// TIA Portal project "Smith Predictor Controller 20211018" (V15.1)

(* hardware
DEVICE "S71500/ET200MP station_1"  S7-1500 station
   slot 0: "导轨_0"  Rack  6ES7 590-1***0-0AA0
   slot 1: "PLC_1"  CPU 1516-3 PN/DP  6ES7 516-3AN01-0AB0  V2.6
      slot 3: "CPU 显示_1"  6ES7591-1BA00-0AA0
*)

// ===== PLC "PLC_1"  CPU 1516-3 PN/DP =====

// folder: smith

DATA_BLOCK "SIM_DB"   // DB1
{ S7_Optimized_Access := 'TRUE' }
VERSION : 0.1
   VAR
      SIM_RUN : Bool;
      PLANT_PV_SMITH : Real;
      PLANT_PV_PID : Real;
      "PLANT_TAU_ACTUAL[ms]" : Real := 500.0;
      "PLANT_DELAY_ACTUAL[Ncycle]" : Int := 50;
      "PLANT_TAU_SET[ms]" : Real := 500.0;
      PLANT_TAU_SET_MIN : Real := 475.0;
      PLANT_TAU_SET_MAX : Real := 525.0;
      "PLANT_DELAY_SET[s]" : Real := 5.0;
      "PLANT_DELAY_SET[Ncycle]" : Int := 50;
      PLANT_DELAY_SET_MIN : Int := 45;
      PLANT_DELAY_SET_MAX : Int := 55;
   END_VAR
BEGIN
END_DATA_BLOCK

DATA_BLOCK "SMITH_DB"   // DB2
{ S7_Optimized_Access := 'TRUE' }
VERSION : 0.1
// stored: InstanceOfName SMITH
"SMITH"
BEGIN
END_DATA_BLOCK

DATA_BLOCK "PID_DB"   // DB3
{ S7_Optimized_Access := 'TRUE' }
VERSION : 0.1
// stored: InstanceOfName PID
"PID"
BEGIN
END_DATA_BLOCK

DATA_BLOCK "LAG1_DB_plant_dummy"   // DB4
{ S7_Optimized_Access := 'TRUE' }
VERSION : 0.1
// stored: InstanceOfName LAG1
"LAG1"
BEGIN
END_DATA_BLOCK

DATA_BLOCK "DELAY_DB_plant_dummy"   // DB5
{ S7_Optimized_Access := 'TRUE' }
VERSION : 0.1
// stored: InstanceOfName DELAY
"DELAY"
BEGIN
END_DATA_BLOCK

DATA_BLOCK "TEST_PID_DB"   // DB6
{ S7_Optimized_Access := 'TRUE' }
VERSION : 0.1
   VAR
      RUN : Bool;
      XIN : Real;
      XOUT : Real;
      X0 : Real;
      KP : Real := 1.0;
      TR : Real := 1000.0;
   END_VAR
BEGIN
END_DATA_BLOCK

DATA_BLOCK "TEST_SMITH_DB"   // DB21
{ S7_Optimized_Access := 'TRUE' }
VERSION : 0.1
   VAR
      RUN : Bool;
      XIN : Real;
      XOUT : Real;
      X0 : Real;
      KP : Real := 0.2;
      TR : Real := 1000.0;
      "PLANT_TAU_PREDICT[ms]" : Real := 500.0;
      "PLANT_DELAY_PREDICT[Ncycle]" : Int := 50;
      "PLANT_DELAY_PREDICT_SET[s]" : Real := 5.0;
      "PLANT_DELAY_PREDICT_SET[Ncycle]" : Int := 50;
      PLANT_DELAY_PREDICT_SET_MIN : Int := 45;
      PLANT_DELAY_PREDICT_SET_MAX : Int := 55;
   END_VAR
BEGIN
END_DATA_BLOCK

DATA_BLOCK "LAG1_DB_plant"   // DB25
{ S7_Optimized_Access := 'TRUE' }
VERSION : 0.1
// stored: InstanceOfName LAG1
"LAG1"
BEGIN
END_DATA_BLOCK

DATA_BLOCK "DELAY_DB_plant"   // DB26
{ S7_Optimized_Access := 'TRUE' }
VERSION : 0.1
// stored: InstanceOfName DELAY
"DELAY"
BEGIN
END_DATA_BLOCK

// folder: (top level)

FUNCTION "LGF_RandomBasic" : Real   // FC10038, SCL
{ S7_Optimized_Access := 'TRUE' }
   VAR_TEMP
      tempTime : DTL;   // System time
      tempTimeStatus : Int;   // Status of the instruction RD_SYS_T
      tempRandomValue : UDInt;   // Random-start-value
   END_VAR
   // Ret_Val : Ret_Val
   VAR CONSTANT
      MIN_UDINT : UDInt := 0;   // UDInt lower value range
      MAX_UDINT : UDInt := 4294967295;   // UDInt upper value range
   END_VAR
BEGIN
   //=============================================================================
   // Siemens AG
   // (c)Copyright 2017
   //-----------------------------------------------------------------------------
   // Library:       LGF (Library General Functions)
   // Tested with:   CPU1212C DC/DC/DC FW:V4.2
   // Engineering:   TIA Portal V14 Upd 1
   // Restrictions:  -
   // Requirements:  PLC (S7-1200 / S7-1500)
   // Functionality: This function generates random numbers. 0.0 <= REAL <= 1.0
   //                (Datatype Real)
   //-----------------------------------------------------------------------------
   // Change log table:
   // Version  Date        In charge/Changes applied
   // 01.00.00 27.01.2017  Siemens Industry Online Support
   //                      First released version
   //-----------------------------------------------------------------------------
   //Status Codes: -
   //=============================================================================

   //Read system time
   #tempTimeStatus := RD_SYS_T(#tempTime);

   //Callculate a random-start-value depending on the time
   #tempRandomValue.%B3 := #tempTime.NANOSECOND.%B0;
   #tempRandomValue.%B2 := #tempTime.NANOSECOND.%B1;
   #tempRandomValue.%B1 := #tempTime.NANOSECOND.%B2;
   #tempRandomValue.%B0 := #tempTime.NANOSECOND.%B3;

   //Norm the calculated random number: 0.0 <= #LGF_RandomBasic <= 1.0
   #LGF_RandomBasic := NORM_X(MIN := #MIN_UDINT, VALUE := #tempRandomValue, MAX := #MAX_UDINT);
END_FUNCTION

ORGANIZATION_BLOCK "Main"   // OB1, LAD, ProgramCycle
TITLE = "Main Program Sweep (Cycle)"
{ S7_Optimized_Access := 'TRUE' }
VERSION : 0.1
   VAR_INPUT
      Initial_Call : Bool;   // Initial call of this OB
      Remanence : Bool;   // =True, if remanent data are available
   END_VAR
BEGIN
END_ORGANIZATION_BLOCK

// folder: smith

FUNCTION_BLOCK "SMITH"   // FB1, LAD
TITLE = Smith Predictor Controller
{ S7_Optimized_Access := 'TRUE' }
VERSION : 0.1
// 2021/10/14 Created by GQ
   VAR_INPUT
      AUTO : Bool;   // 0 - manual , 1 - automatic
      "PLANT_TAU[ms]" : Real;
      "PLANT_DELAY[Ncycle]" : Int;
      DBW : Real;   // Deadband Width
      SP : Real;   // Set point
      PV : Real;   // Process variable
      X0 : Real;   // Manual output adjustment
      KP : Real;   // Proportionality constant
      "TR[ms]" : Real;   // Reset time
      "TD[ms]" : Real;   // Derivative time constant
      RATEVALUE : Real;   // value change limiter for every cycle
      MN : Real;
      MX : Real;
      "CYCLE[ms]" : Real;   // Sampling period
   END_VAR
   VAR_OUTPUT
      XOUT : Real;
      STATUSINFO : Word;
   END_VAR
   VAR
      Y0 : Real;   // Predicted Output
      Y1 : Real;   // Predicted Output with Delay
      ERROR : Real;   // SP-PV
      E0 : Real;   // ERROR for PID
      E0DBW : Real;   // E0 with Deadband
      PIDOUT : Real;
      ITERM : "INTEGRAL";
      DTERM : "DERIVATIVE";
      PLANT : "LAG1";   // Plant Model
      PLANTDELAY : "DELAY";
      RATELIMITER : "RateLimiter";
   END_VAR
   VAR CONSTANT
      NO_ERROR : Word := 16#0000;   // No errors
      I_TIME : Word := 16#7000;   // Integral time constant error
      OUT_ARRAY_INDEX : Word := 16#8000;   // Index out of array range
      LIMIT_PARA_FAULT : Word := 16#8200;   // MAX less then MIN in limit
      RATEVALUE_ZERO : Word := 16#8400;   // Rate value zero
   END_VAR
BEGIN

REGION Network 1 (SCL): License
   //=============================================================================
   // (c)Copyright 2021
   //-----------------------------------------------------------------------------
   // Library:       
   // Tested with:   PLCSim Advanced
   // Engineering:   TIA Portal V15 Update 1
   // Restrictions:  
   // Requirements:  PLC (S7-1200 / S7-1500)
   // Functionality: Smith Predictor Controller
   //-----------------------------------------------------------------------------
   // Change log table:
   // Version  Date        In charge / Changes applied
   // 00.00.01 10.14.2021  002706      created
   //=============================================================================


   IF #"TR[ms]" <= 0.0 THEN
       #STATUSINFO := #I_TIME;
       RETURN;
   END_IF;

   IF #"PLANT_DELAY[Ncycle]" > 127 OR #"PLANT_DELAY[Ncycle]" < 0 THEN
       #STATUSINFO := #OUT_ARRAY_INDEX;
       RETURN;
   END_IF;

   IF #MX < #MN THEN
       #STATUSINFO := #LIMIT_PARA_FAULT;
       RETURN
       ;
   END_IF;

   IF #RATEVALUE = 0.0 OR #RATEVALUE > (#MX - #MN)THEN
       #STATUSINFO := #RATEVALUE_ZERO;
       RETURN
       ;
   END_IF;

   #STATUSINFO := #NO_ERROR;
END_REGION

REGION Network 2: Y0
   // Output of predicted plant model
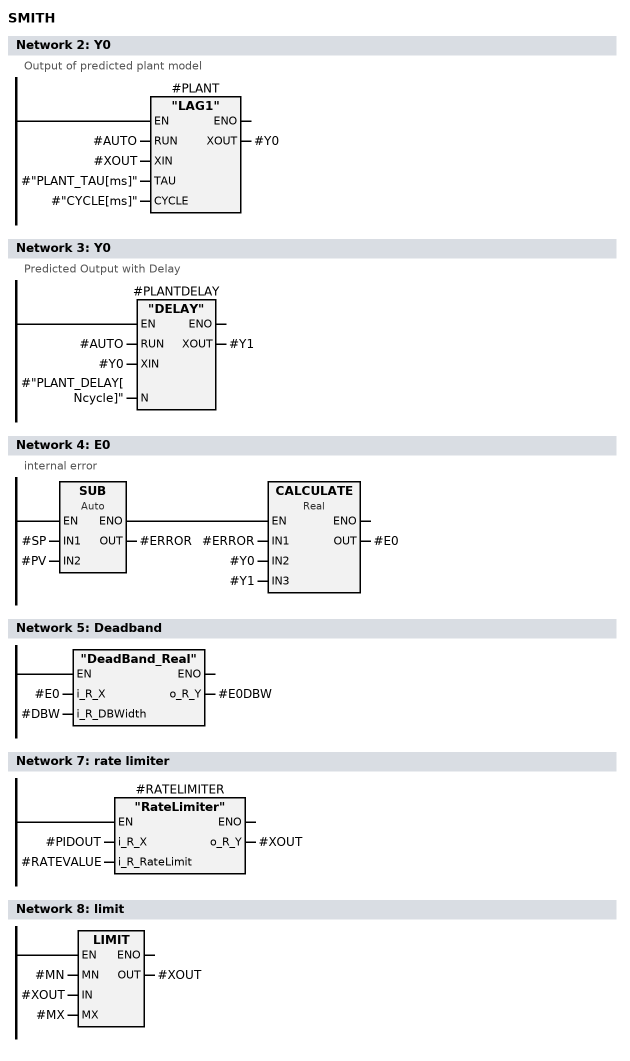
   RUNG wire#powerrail
      #PLANT(RUN := #AUTO, XIN := #XOUT, TAU := #"PLANT_TAU[ms]", CYCLE := #"CYCLE[ms]", XOUT => #Y0)
   END_RUNG
   // the same network as SCL:
   #PLANT(RUN := #AUTO, XIN := #XOUT, TAU := #"PLANT_TAU[ms]", CYCLE := #"CYCLE[ms]", XOUT => #Y0);   // "LAG1"
END_REGION

REGION Network 3: Y0
   // Predicted Output with Delay
   RUNG wire#powerrail
      #PLANTDELAY(RUN := #AUTO, XIN := #Y0, N := #"PLANT_DELAY[Ncycle]", XOUT => #Y1)
   END_RUNG
   // the same network as SCL:
   #PLANTDELAY(RUN := #AUTO, XIN := #Y0, N := #"PLANT_DELAY[Ncycle]", XOUT => #Y1);   // "DELAY"
END_REGION

REGION Network 4: E0
   // internal error
   RUNG wire#powerrail
      Sub(in1 := #SP, in2 := #PV, out => #ERROR)
      { S7_Templates := "SrcType := Real"; S7_Expression := "IN1 - (IN2 - IN3)" } Calculate(in1 := #ERROR, in2 := #Y0, in3 := #Y1, out => #E0)
   END_RUNG
   // the same network as SCL:
   #ERROR := #SP - #PV;
   #E0 := #ERROR - (#Y0 - #Y1);
END_REGION

REGION Network 5: Deadband
   RUNG wire#powerrail
      "DeadBand_Real"(i_R_X := #E0, i_R_DBWidth := #DBW, o_R_Y => #E0DBW)
   END_RUNG
   // the same network as SCL:
   "DeadBand_Real"(i_R_X := #E0, i_R_DBWidth := #DBW, o_R_Y => #E0DBW);
END_REGION

REGION Network 6 (SCL): PID
   // https://blog.opticontrols.com/archives/383
   // The Cohen-Coon tuning rules were designed for controllers with the noninteractive controller algorithm.
   // Different PID algorithm  equation will cause different result.
   // PID
   (*** Adjust ITERM so that XOUT := X0 when AUTO = 0 ***)
   IF #KP = 0.0 THEN
       #PIDOUT := 0.0;
   ELSE
       #ITERM(RUN := #AUTO,
              R1 := NOT #AUTO,
              XIN := #E0DBW,
              X0 := #"TR[ms]" * (#X0 / #KP - #E0DBW),
              CYCLE := #"CYCLE[ms]");
       #DTERM(RUN := #AUTO,
              XIN := #E0DBW,
              CYCLE := #"CYCLE[ms]");
       #PIDOUT := #KP * (#E0DBW + #ITERM.XOUT / #"TR[ms]" + #DTERM.XOUT * #"TD[ms]");
   END_IF;
END_REGION

REGION Network 7: rate limiter
   RUNG wire#powerrail
      #RATELIMITER(i_R_X := #PIDOUT, i_R_RateLimit := #RATEVALUE, o_R_Y => #XOUT)
   END_RUNG
   // the same network as SCL:
   #RATELIMITER(i_R_X := #PIDOUT, i_R_RateLimit := #RATEVALUE, o_R_Y => #XOUT);   // "RateLimiter"
END_REGION

REGION Network 8: limit
   #XOUT := LIMIT(MN := #MN, IN := #XOUT, MX := #MX);
END_REGION
END_FUNCTION_BLOCK

FUNCTION_BLOCK "DELAY"   // FB2, LAD
{ S7_Optimized_Access := 'TRUE' }
VERSION : 0.1
   VAR_INPUT
      RUN : Bool;   // 1 = run, 0 = reset
      XIN : Real;
      N : Int;   // 0 <= N < 128 or specified maximum value
   END_VAR
   VAR_OUTPUT
      XOUT : Real;   // Delayed output
   END_VAR
   VAR
      X : Array[0..127] of Real;   // N-Element queue with FIFO discipline
      I : Int;
      ID : Int;
   END_VAR
BEGIN

REGION Network 1 (SCL)
   IF #RUN THEN
       FOR #ID := 127 TO 1 BY -1 DO
           #X[#ID] := #X[#ID - 1];
       END_FOR;
       #X[0] := #XIN;
       #XOUT := #X[#N];
   ELSE
       #XOUT := #XIN;
       FOR #I := 0 TO #N DO
           #X[#I] := #XIN;
       END_FOR;
   END_IF;
END_REGION
END_FUNCTION_BLOCK

FUNCTION_BLOCK "LAG1"   // FB3, LAD
{ S7_Optimized_Access := 'TRUE' }
VERSION : 0.1
   VAR_INPUT
      RUN : Bool;
      XIN : Real;
      TAU : Real;
      CYCLE : Real;
   END_VAR
   VAR_OUTPUT
      XOUT : Real;
   END_VAR
   VAR
      K : Real;
   END_VAR
BEGIN

REGION Network 1 (SCL)
   IF #RUN THEN
       #XOUT := #XOUT + #K * (#XIN - #XOUT);
   ELSE
       #XOUT := #XIN;
       #K := #CYCLE / (#CYCLE + #TAU);
   END_IF;
END_REGION
END_FUNCTION_BLOCK

FUNCTION_BLOCK "INTEGRAL"   // FB5, LAD
{ S7_Optimized_Access := 'TRUE' }
VERSION : 0.1
   VAR_INPUT
      RUN : Bool;   // 1 = integrate, 0 = hold
      R1 : Bool;   // Overriding reset
      XIN : Real;   // Input variable
      X0 : Real;   // Initial value
      CYCLE : Real;   // Sampling period
   END_VAR
   VAR_OUTPUT
      Q : Bool;   // NOT R1
      XOUT : Real;   // Integrated output
   END_VAR
BEGIN

REGION Network 1 (SCL): NOT R1
   #Q := NOT #R1;
   IF #R1 THEN #XOUT := #X0;
   ELSIF #RUN THEN
       #XOUT := #XOUT + #XIN *#CYCLE;
   END_IF;
END_REGION
END_FUNCTION_BLOCK

FUNCTION_BLOCK "DERIVATIVE"   // FB6, LAD
{ S7_Optimized_Access := 'TRUE' }
VERSION : 0.1
   VAR_INPUT
      RUN : Bool;   // 0 = reset
      XIN : Real;   // Input to be differentiated
      CYCLE : Real;   // Sampling period
   END_VAR
   VAR_OUTPUT
      XOUT : Real;   // Differentiated output
   END_VAR
   VAR
      X1 : Real;
      X2 : Real;
      X3 : Real;
   END_VAR
BEGIN

REGION Network 1 (SCL): Differentiated output
   IF #RUN THEN
       #XOUT := (3.0 * (#XIN - #X3) + #X1 - #X2) / (10.0 * #CYCLE);
       #X3 := #X2;
       #X2 := #X1;
       #X1 := #XIN;
   ELSE
       #XOUT := 0.0;
       #X1 := #XIN;
       #X2 := #XIN;
       #X3 := #XIN;
   END_IF;
END_REGION
END_FUNCTION_BLOCK

FUNCTION_BLOCK "RateLimiter"   // FB9, SCL
{ S7_Optimized_Access := 'TRUE' }
VERSION : 0.1
   VAR_INPUT
      i_R_X : Real;
      i_R_RateLimit : Real;
   END_VAR
   VAR_OUTPUT
      o_R_Y : Real;
   END_VAR
   VAR
      s_R_Y : Real;
      s_R_B4Y : Real;
   END_VAR
   VAR_TEMP
      t_R_Diff : Real;
      t_R_AbsDiff : Real;
      t_R_AbsRateLimit : Real;
      t_R_MinusRateLimit : Real;
   END_VAR
BEGIN

   // Difference = IN - Yn-1
   #t_R_Diff := (#i_R_X - #s_R_B4Y);
   #t_R_AbsDiff := ABS(#t_R_Diff);
   #t_R_AbsRateLimit := ABS(#i_R_RateLimit);
   #t_R_MinusRateLimit := (-1.0) * #i_R_RateLimit;
   // When +|D| ≥ Difference ≥ –|D|: Y = IN
   // When +|D| < Difference: Y = Yn-1 + |D|
   // When –|D| > Difference: Y = Yn-1 - |D|
   IF
       #t_R_AbsDiff <= #t_R_AbsRateLimit
   THEN
       #s_R_Y := #i_R_X;
   ELSIF
       #t_R_AbsRateLimit < #t_R_Diff
   THEN
       #s_R_Y := #s_R_B4Y + #t_R_AbsRateLimit;
   ELSIF
       #t_R_Diff < #t_R_MinusRateLimit
   THEN
       #s_R_Y := #s_R_B4Y - #t_R_AbsRateLimit;
   ELSE
       #s_R_Y := #i_R_X;
   END_IF;
   #s_R_B4Y := #s_R_Y;

   #o_R_Y := #s_R_Y;
END_FUNCTION_BLOCK

FUNCTION_BLOCK "PID"   // FB10, LAD
TITLE = PID Controller
{ S7_Optimized_Access := 'TRUE' }
VERSION : 0.1
// 2021/10/14 Created by GQ
   VAR_INPUT
      AUTO : Bool;   // 0 - manual , 1 - automatic
      DBW : Real;   // Deadband Width
      SP : Real;   // Set point
      PV : Real;   // Process variable
      X0 : Real;   // Manual output adjustment
      KP : Real;   // Proportionality constant
      "TR[ms]" : Real;   // Reset time
      "TD[ms]" : Real;   // Derivative time constant
      RATEVALUE : Real;   // value change limiter for every cycle
      MN : Real;
      MX : Real;
      "CYCLE[ms]" : Real;   // Sampling period
   END_VAR
   VAR_OUTPUT
      XOUT : Real;
      STATUSINFO : Word;
   END_VAR
   VAR
      ERROR : Real;   // SP-PV
      EDBW : Real;   // ERROR with Deadband
      PIDOUT : Real;
      ITERM : "INTEGRAL";
      DTERM : "DERIVATIVE";
      RATELIMITER : "RateLimiter";
   END_VAR
   VAR CONSTANT
      NO_ERROR : Word := 16#0000;   // No errors
      I_TIME : Word := 16#7000;   // Integral time constant error
      OUT_ARRAY_INDEX : Word := 16#8000;   // Index out of array range
      LIMIT_PARA_FAULT : Word := 16#8200;   // MAX less then MIN in limit
      RATEVALUE_ZERO : Word := 16#8400;   // Rate value zero
   END_VAR
BEGIN

REGION Network 1 (SCL): License
   //=============================================================================
   // (c)Copyright 2021
   //-----------------------------------------------------------------------------
   // Library:       
   // Tested with:   PLCSim Advanced
   // Engineering:   TIA Portal V15 Update 1
   // Restrictions:  
   // Requirements:  PLC (S7-1200 / S7-1500)
   // Functionality: PID Controller for check result of smith predictor
   //-----------------------------------------------------------------------------
   // Change log table:
   // Version  Date        In charge / Changes applied
   // 00.00.01 10.14.2021  002706      created
   //=============================================================================


   IF #"TR[ms]" <= 0.0 THEN
       #STATUSINFO := #I_TIME;
       RETURN;
   END_IF;

   IF #MX < #MN THEN
       #STATUSINFO := #LIMIT_PARA_FAULT;
       RETURN
       ;
   END_IF;

   IF #RATEVALUE = 0.0 OR #RATEVALUE > (#MX - #MN)THEN
       #STATUSINFO := #RATEVALUE_ZERO;
       RETURN
       ;
   END_IF;

   #STATUSINFO := #NO_ERROR;
END_REGION

REGION Network 2: ERROR
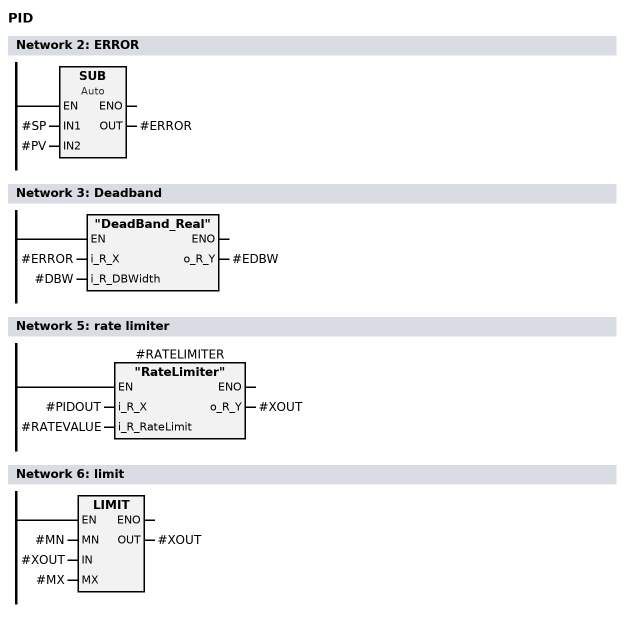
   RUNG wire#powerrail
      Sub(in1 := #SP, in2 := #PV, out => #ERROR)
   END_RUNG
   // the same network as SCL:
   #ERROR := #SP - #PV;
END_REGION

REGION Network 3: Deadband
   RUNG wire#powerrail
      "DeadBand_Real"(i_R_X := #ERROR, i_R_DBWidth := #DBW, o_R_Y => #EDBW)
   END_RUNG
   // the same network as SCL:
   "DeadBand_Real"(i_R_X := #ERROR, i_R_DBWidth := #DBW, o_R_Y => #EDBW);
END_REGION

REGION Network 4 (SCL): PID
   // https://blog.opticontrols.com/archives/383
   // The Cohen-Coon tuning rules were designed for controllers with the noninteractive controller algorithm.
   // Different PID algorithm  equation will cause different result.
   // PID
   (*** Adjust ITERM so that XOUT := X0 when AUTO = 0 ***)
   IF #KP = 0.0 THEN
       #PIDOUT := 0.0;
   ELSE
       #ITERM(RUN := #AUTO,
              R1 := NOT #AUTO,
              XIN := #EDBW,
              X0 := #"TR[ms]" * (#X0 - #EDBW),
              CYCLE := #"CYCLE[ms]");
       #DTERM(RUN := #AUTO,
              XIN := #EDBW,
              CYCLE := #"CYCLE[ms]");
       #PIDOUT := #KP * (#EDBW + #ITERM.XOUT / #"TR[ms]" + #DTERM.XOUT * #"TD[ms]");
   END_IF;
END_REGION

REGION Network 5: rate limiter
   RUNG wire#powerrail
      #RATELIMITER(i_R_X := #PIDOUT, i_R_RateLimit := #RATEVALUE, o_R_Y => #XOUT)
   END_RUNG
   // the same network as SCL:
   #RATELIMITER(i_R_X := #PIDOUT, i_R_RateLimit := #RATEVALUE, o_R_Y => #XOUT);   // "RateLimiter"
END_REGION

REGION Network 6: limit
   #XOUT := LIMIT(MN := #MN, IN := #XOUT, MX := #MX);
END_REGION
END_FUNCTION_BLOCK

FUNCTION "LGF_RandomInt" : Int   // FC10013, SCL
{ S7_Optimized_Access := 'TRUE' }
   VAR_INPUT
      minValue : Int;   // minimal Value random can reach
      maxValue : Int;   // maximal Value random can reach
   END_VAR
   VAR_OUTPUT
      error : Bool;
      statusID : UInt;
      status : Word;
   END_VAR
   VAR_TEMP
      tempTime : DTL;
      tempTimeStatus : Int;
      tempRandomValue : Int;
      tempNormReal : Real;
   END_VAR
   VAR CONSTANT
      NO_ERROR : Word := 16#0000;
      NO_CURRENT_JOBS : Word := 16#7000;
      MAX_LESS_MIN : Word := 16#8200;
      ERROR_IN_THIS_BLOCK : UInt := 1;
      ERROR_RD_SYS_T : UInt := 2;
      MIN_INT : DInt := -32768;
      MAX_INT : DInt := 32767;
   END_VAR
BEGIN
   //=============================================================================
   // Siemens AG
   // (c)Copyright 2017
   //-----------------------------------------------------------------------------
   // Library:       LGF (Library General Functions)
   // Tested with:   CPU1212C DC/DC/DC FW:V4.2
   // Engineering:   TIA Portal V13 SP1 Upd 4
   // Restrictions:  -
   // Requirements:  PLC (S7-1200 / S7-1500)
   // Functionality: This function generates random numbers in defined limits
   //                (Datatype Int)
   //-----------------------------------------------------------------------------
   // Change log table:
   // Version  Date        In charge / Changes applied
   // 01.00.00 19.08.2015  Siemens Industry Online Support
   //                      First released version
   // 01.00.01 02.01.2017  Siemens Industry Online Support
   //                      Upgrade: TIA Portal V14 Update 1
   // 01.00.01 10.18.2021  Scale_X 替换成公式 OUT = [VALUE ∗ (MAX – MIN)] + MIN                    
   //-----------------------------------------------------------------------------
   //Status Codes:
   // 16#7000:  No current jobs
   // 16#0000:  Job finished; Note: There is no "Busy"-Status because the block
   //           is finished within a single cycle
   // 16#8200:  maxValue is samller then minValue 
   //=============================================================================

   //Set "No current job" status
   #error := false;
   #statusID := #ERROR_IN_THIS_BLOCK;
   #status := #NO_CURRENT_JOBS;

   //Check if the maximal Value is less than the minimal value
   IF (#minValue > #maxValue) THEN
     #error := true;
     #statusID := #ERROR_IN_THIS_BLOCK;
     #status := #MAX_LESS_MIN;
     #LGF_RandomInt := 0;
     RETURN;
   END_IF;

   //Read system time
   #tempTimeStatus := RD_SYS_T(#tempTime);

   IF (#tempTimeStatus <> 0) THEN
     #error := true;
     #statusID := #ERROR_RD_SYS_T;
     #status := INT_TO_WORD(#tempTimeStatus);
     #LGF_RandomInt := 0;
     RETURN;
   END_IF;

   //Callculate a random-start-value depending on the time
   #tempRandomValue.%B1 := #tempTime.NANOSECOND.%B0;
   #tempRandomValue.%B0 := #tempTime.NANOSECOND.%B1;

   //adapt the calculated random number to the given number span
   #tempNormReal := NORM_X(MIN := #MIN_INT, VALUE := #tempRandomValue, MAX := #MAX_INT);
   // #LGF_RandomInt := SCALE_X(MIN := #minValue, VALUE := #tempNormReal, MAX := #maxValue);
   #LGF_RandomInt := REAL_TO_INT(#tempNormReal * (#maxValue - #minValue) + #minValue);

   #status := #NO_ERROR;
END_FUNCTION

FUNCTION "LGF_RandomReal" : Real   // FC10014, SCL
{ S7_Optimized_Access := 'TRUE' }
   VAR_INPUT
      minValue : Real;   // minimal Value random can reach
      maxValue : Real;   // maximal Value random can reach
   END_VAR
   VAR_OUTPUT
      error : Bool;
      statusID : UInt;
      status : Word;
   END_VAR
   VAR_TEMP
      tempTime : DTL;
      tempTimeStatus : Int;
      tempRandomValue : UDInt;
      tempNormReal : Real;
   END_VAR
   VAR CONSTANT
      NO_ERROR : Word := 16#0000;
      NO_CURRENT_JOBS : Word := 16#7000;
      MAX_LESS_MIN : Word := 16#8200;
      ERROR_IN_THIS_BLOCK : UInt := 1;
      ERROR_RD_SYS_T : UInt := 2;
      MIN_UDINT : UDInt := 0;
      MAX_UDINT : UDInt := 4294967295;
   END_VAR
BEGIN
   //=============================================================================
   // Siemens AG
   // (c)Copyright 2017
   //-----------------------------------------------------------------------------
   // Library:       LGF (Library General Functions)
   // Tested with:   CPU1212C DC/DC/DC FW:V4.2
   // Engineering:   TIA Portal V14 Update 1
   // Restrictions:  -
   // Requirements:  PLC (S7-1200 / S7-1500)
   // Functionality: This function generates random numbers in defined limits
   //                (Datatype Real)
   //-----------------------------------------------------------------------------
   // Change log table:
   // Version  Date        In charge / Changes applied
   // 01.00.00 19.08.2015  Siemens Industry Online Support
   //                      First released version
   // 01.00.01 02.01.2017  Siemens Industry Online Support
   //                      Upgrade: TIA Portal V14 Update 1
   // 01.00.02 02.03.2017  Siemens Industry Online Support
   //                      Bugfix: FC number
   // 01.00.01 10.18.2021  Scale_X 替换成公式 OUT = [VALUE ∗ (MAX – MIN)] + MIN       
   //-----------------------------------------------------------------------------
   //Status Codes:
   // 16#7000:  No current jobs
   // 16#0000:  Job finished   // Note: There is no "Busy"-Status because the
   //           block is finished within a single cycle
   // 16#8200:  maxValue is samller then minValue 
   //=============================================================================

   //Set "No current job" status
   #error := false;
   #statusID := #ERROR_IN_THIS_BLOCK;
   #status := #NO_CURRENT_JOBS;

   //Check if the maximal Value is less than the minimal value
   IF (#minValue > #maxValue) THEN
     #error := true;
     #statusID := #ERROR_IN_THIS_BLOCK;
     #status := #MAX_LESS_MIN;
     #LGF_RandomReal := 0;
     RETURN;
   END_IF;

   //Read system time
   #tempTimeStatus := RD_SYS_T(#tempTime);

   IF (#tempTimeStatus <> 0) THEN
     #error := true;
     #statusID := #ERROR_RD_SYS_T;
     #status := INT_TO_WORD(#tempTimeStatus);
     #LGF_RandomReal := 0;
     RETURN;
   END_IF;

   //Callculate a random-start-value depending on the time
   #tempRandomValue.%B3 := #tempTime.NANOSECOND.%B0;
   #tempRandomValue.%B2 := #tempTime.NANOSECOND.%B1;
   #tempRandomValue.%B1 := #tempTime.NANOSECOND.%B2;
   #tempRandomValue.%B0 := #tempTime.NANOSECOND.%B3;

   //adapt the calculated random number to the given number span
   #tempNormReal := NORM_X(MIN := #MIN_UDINT, VALUE := #tempRandomValue, MAX := #MAX_UDINT);
   // #LGF_RandomReal := SCALE_X(MIN := #minValue, VALUE := #tempNormReal, MAX := #maxValue);
   #LGF_RandomReal := #tempNormReal * (#maxValue - #minValue) + #minValue;

   #status := #NO_ERROR;
END_FUNCTION

FUNCTION "DeadBand_Real" : Void   // FC30005, SCL
{ S7_Optimized_Access := 'TRUE' }
VERSION : 0.1
   VAR_INPUT
      i_R_X : Real;
      i_R_DBWidth : Real;
   END_VAR
   VAR_OUTPUT
      o_R_Y : Real;
   END_VAR
   VAR_TEMP
      i_R_AbsX : Real;
      i_R_AbsDBWidth : Real;
   END_VAR
BEGIN
   #i_R_AbsX := ABS(#i_R_X);
   #i_R_AbsDBWidth := ABS(#i_R_DBWidth);
   IF #i_R_AbsX > #i_R_AbsDBWidth AND #i_R_X >= 0 THEN
       #o_R_Y := #i_R_X - #i_R_AbsDBWidth;
   ELSIF #i_R_AbsX > #i_R_AbsDBWidth AND #i_R_X < 0 THEN
       #o_R_Y := #i_R_X + #i_R_AbsDBWidth;
   ELSE
       #o_R_Y := REAL#0.0;
   END_IF;
END_FUNCTION

ORGANIZATION_BLOCK "Cyclic interrupt"   // OB30, LAD, CyclicInterrupt
TITLE = Smith控制器
{ S7_Optimized_Access := 'TRUE' }
VERSION : 0.1
   VAR_INPUT
      Initial_Call : Bool;   // Initial call of this OB
      Event_Count : Int;   // Events discarded
   END_VAR
   VAR_TEMP
      dy : Real;
      yp : Real;
      y1 : Real;
      dp : Real;
      ya : Real;
      TEMP1 : Bool;
      TEMP2 : UInt;
      TEMP3 : Word;
   END_VAR
BEGIN

REGION Network 1 (SCL): 延时时间设定
   "TEST_SMITH_DB"."PLANT_DELAY_PREDICT_SET[Ncycle]" := "TEST_SMITH_DB"."PLANT_DELAY_PREDICT_SET[s]" * 1000.0 / 100.0;
   "TEST_SMITH_DB".PLANT_DELAY_PREDICT_SET_MIN := "TEST_SMITH_DB"."PLANT_DELAY_PREDICT_SET[Ncycle]" * 0.80;
   "TEST_SMITH_DB".PLANT_DELAY_PREDICT_SET_MAX := "TEST_SMITH_DB"."PLANT_DELAY_PREDICT_SET[Ncycle]" * 1.2;
END_REGION

REGION Network 2: 实际延时时间
   // 0.8~1.2，设置+/-20%用于跟踪不准确
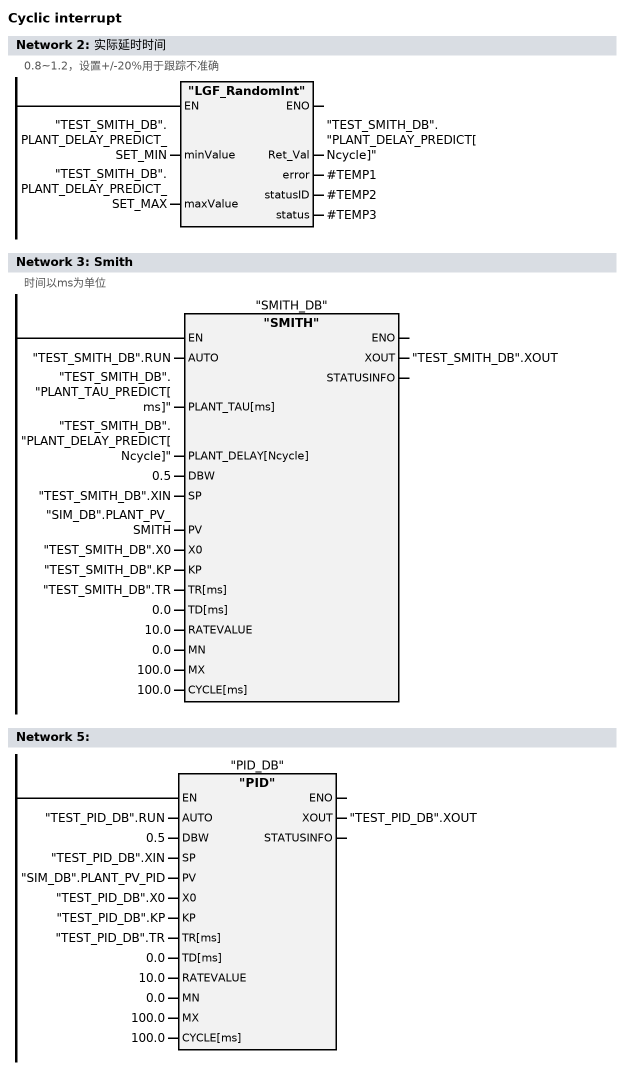
   RUNG wire#powerrail
      "LGF_RandomInt"(minValue := "TEST_SMITH_DB".PLANT_DELAY_PREDICT_SET_MIN, maxValue := "TEST_SMITH_DB".PLANT_DELAY_PREDICT_SET_MAX, Ret_Val => "TEST_SMITH_DB"."PLANT_DELAY_PREDICT[Ncycle]", error => #TEMP1, statusID => #TEMP2, status => #TEMP3)
   END_RUNG
   // the same network as SCL:
   "TEST_SMITH_DB"."PLANT_DELAY_PREDICT[Ncycle]" := "LGF_RandomInt"(minValue := "TEST_SMITH_DB".PLANT_DELAY_PREDICT_SET_MIN,
                           maxValue := "TEST_SMITH_DB".PLANT_DELAY_PREDICT_SET_MAX,
                           error => #TEMP1,
                           statusID => #TEMP2,
                           status => #TEMP3);
END_REGION

REGION Network 3: Smith
   // 时间以ms为单位
   RUNG wire#powerrail
      "SMITH_DB"(AUTO := "TEST_SMITH_DB".RUN, "PLANT_TAU[ms]" := "TEST_SMITH_DB"."PLANT_TAU_PREDICT[ms]", "PLANT_DELAY[Ncycle]" := "TEST_SMITH_DB"."PLANT_DELAY_PREDICT[Ncycle]", DBW := 0.5, SP := "TEST_SMITH_DB".XIN, PV := "SIM_DB".PLANT_PV_SMITH, X0 := "TEST_SMITH_DB".X0, KP := "TEST_SMITH_DB".KP, "TR[ms]" := "TEST_SMITH_DB".TR, "TD[ms]" := 0.0, RATEVALUE := 10.0, MN := 0.0, MX := 100.0, "CYCLE[ms]" := 100.0, XOUT => "TEST_SMITH_DB".XOUT, STATUSINFO =>)
   END_RUNG
   // the same network as SCL:
   "SMITH_DB"(AUTO := "TEST_SMITH_DB".RUN,   // "SMITH"
              "PLANT_TAU[ms]" := "TEST_SMITH_DB"."PLANT_TAU_PREDICT[ms]",
              "PLANT_DELAY[Ncycle]" := "TEST_SMITH_DB"."PLANT_DELAY_PREDICT[Ncycle]",
              DBW := 0.5,
              SP := "TEST_SMITH_DB".XIN,
              PV := "SIM_DB".PLANT_PV_SMITH,
              X0 := "TEST_SMITH_DB".X0,
              KP := "TEST_SMITH_DB".KP,
              "TR[ms]" := "TEST_SMITH_DB".TR,
              "TD[ms]" := 0.0,
              RATEVALUE := 10.0,
              MN := 0.0,
              MX := 100.0,
              "CYCLE[ms]" := 100.0,
              XOUT => "TEST_SMITH_DB".XOUT);
END_REGION

REGION Network 4 (SCL)
   "TEST_PID_DB".RUN := "TEST_SMITH_DB".RUN;
   "TEST_PID_DB".XIN := "TEST_SMITH_DB".XIN;
   "TEST_PID_DB".X0 := "TEST_SMITH_DB".X0;
   "TEST_PID_DB".KP := "TEST_SMITH_DB".KP;
   "TEST_PID_DB".TR := "TEST_SMITH_DB".TR;
END_REGION

REGION Network 5
   RUNG wire#powerrail
      "PID_DB"(AUTO := "TEST_PID_DB".RUN, DBW := 0.5, SP := "TEST_PID_DB".XIN, PV := "SIM_DB".PLANT_PV_PID, X0 := "TEST_PID_DB".X0, KP := "TEST_PID_DB".KP, "TR[ms]" := "TEST_PID_DB".TR, "TD[ms]" := 0.0, RATEVALUE := 10.0, MN := 0.0, MX := 100.0, "CYCLE[ms]" := 100.0, XOUT => "TEST_PID_DB".XOUT, STATUSINFO =>)
   END_RUNG
   // the same network as SCL:
   "PID_DB"(AUTO := "TEST_PID_DB".RUN,   // "PID"
            DBW := 0.5,
            SP := "TEST_PID_DB".XIN,
            PV := "SIM_DB".PLANT_PV_PID,
            X0 := "TEST_PID_DB".X0,
            KP := "TEST_PID_DB".KP,
            "TR[ms]" := "TEST_PID_DB".TR,
            "TD[ms]" := 0.0,
            RATEVALUE := 10.0,
            MN := 0.0,
            MX := 100.0,
            "CYCLE[ms]" := 100.0,
            XOUT => "TEST_PID_DB".XOUT);
END_REGION
END_ORGANIZATION_BLOCK

ORGANIZATION_BLOCK "Cyclic interrupt_sim"   // OB31, LAD, CyclicInterrupt
TITLE = 仿真测试
{ S7_Optimized_Access := 'TRUE' }
VERSION : 0.1
   VAR_INPUT
      Initial_Call : Bool;   // Initial call of this OB
      Event_Count : Int;   // Events discarded
   END_VAR
   VAR_TEMP
      TEMP1 : Bool;
      TEMP2 : UInt;
      TEMP3 : Word;
      TEMP4 : Bool;
      TEMP5 : UInt;
      TEMP6 : Word;
   END_VAR
   VAR CONSTANT
      CYCLE : Real := 100.0;   // 扫描周期100ms
   END_VAR
   VAR_TEMP   // added for the SCL form of the ladder/FBD networks
      _w1 : Bool;
   END_VAR
BEGIN

REGION Network 1 (SCL)
   "SIM_DB".PLANT_TAU_SET_MIN := "SIM_DB"."PLANT_TAU_SET[ms]" * 0.95;
   "SIM_DB".PLANT_TAU_SET_MAX := "SIM_DB"."PLANT_TAU_SET[ms]" * 1.05;

   "SIM_DB"."PLANT_DELAY_SET[Ncycle]" := "SIM_DB"."PLANT_DELAY_SET[s]" * 1000.0 / #CYCLE;
   "SIM_DB".PLANT_DELAY_SET_MIN := "SIM_DB"."PLANT_DELAY_SET[Ncycle]" * 0.95;
   "SIM_DB".PLANT_DELAY_SET_MAX := "SIM_DB"."PLANT_DELAY_SET[Ncycle]" * 1.05;
END_REGION

REGION Network 2: 实际时间常数
   // 0.95~1.05
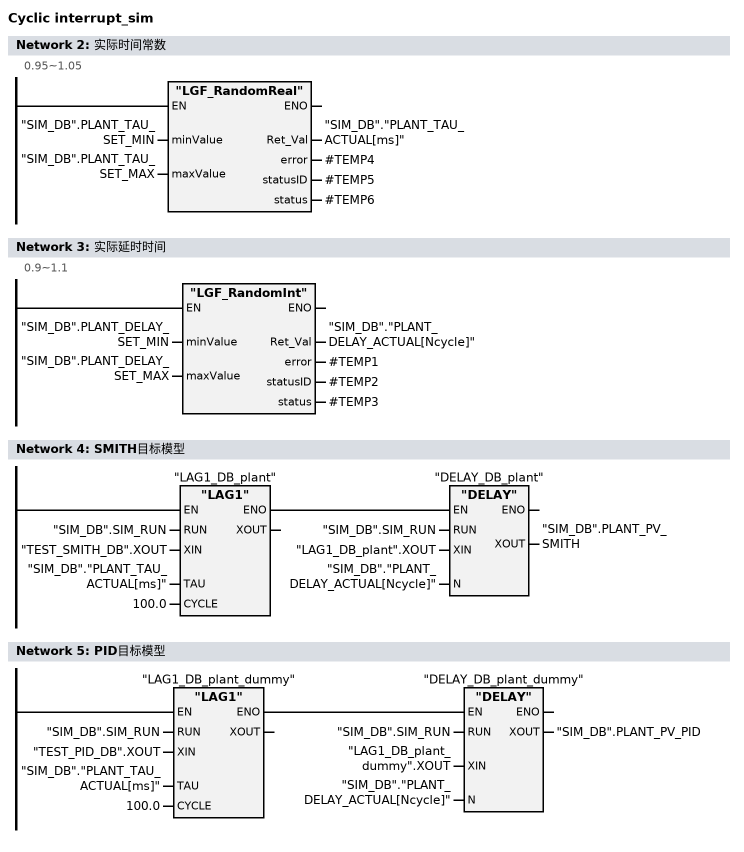
   RUNG wire#powerrail
      "LGF_RandomReal"(minValue := "SIM_DB".PLANT_TAU_SET_MIN, maxValue := "SIM_DB".PLANT_TAU_SET_MAX, Ret_Val => "SIM_DB"."PLANT_TAU_ACTUAL[ms]", error => #TEMP4, statusID => #TEMP5, status => #TEMP6)
   END_RUNG
   // the same network as SCL:
   "SIM_DB"."PLANT_TAU_ACTUAL[ms]" := "LGF_RandomReal"(minValue := "SIM_DB".PLANT_TAU_SET_MIN,
                           maxValue := "SIM_DB".PLANT_TAU_SET_MAX,
                           error => #TEMP4,
                           statusID => #TEMP5,
                           status => #TEMP6);
END_REGION

REGION Network 3: 实际延时时间
   // 0.9~1.1
   RUNG wire#powerrail
      "LGF_RandomInt"(minValue := "SIM_DB".PLANT_DELAY_SET_MIN, maxValue := "SIM_DB".PLANT_DELAY_SET_MAX, Ret_Val => "SIM_DB"."PLANT_DELAY_ACTUAL[Ncycle]", error => #TEMP1, statusID => #TEMP2, status => #TEMP3)
   END_RUNG
   // the same network as SCL:
   "SIM_DB"."PLANT_DELAY_ACTUAL[Ncycle]" := "LGF_RandomInt"(minValue := "SIM_DB".PLANT_DELAY_SET_MIN,
                           maxValue := "SIM_DB".PLANT_DELAY_SET_MAX,
                           error => #TEMP1,
                           statusID => #TEMP2,
                           status => #TEMP3);
END_REGION

REGION Network 4: SMITH目标模型
   RUNG wire#powerrail
      "LAG1_DB_plant"(RUN := "SIM_DB".SIM_RUN, XIN := "TEST_SMITH_DB".XOUT, TAU := "SIM_DB"."PLANT_TAU_ACTUAL[ms]", CYCLE := 100.0, XOUT =>)
      "DELAY_DB_plant"(RUN := "SIM_DB".SIM_RUN, XIN := "LAG1_DB_plant".XOUT, N := "SIM_DB"."PLANT_DELAY_ACTUAL[Ncycle]", XOUT => "SIM_DB".PLANT_PV_SMITH)
   END_RUNG
   // the same network as SCL:
   "LAG1_DB_plant"(RUN := "SIM_DB".SIM_RUN,   // "LAG1"
                   XIN := "TEST_SMITH_DB".XOUT,
                   TAU := "SIM_DB"."PLANT_TAU_ACTUAL[ms]",
                   CYCLE := 100.0,
                   ENO => #_w1);
   IF #_w1 THEN
       "DELAY_DB_plant"(RUN := "SIM_DB".SIM_RUN,   // "DELAY"
                        XIN := "LAG1_DB_plant".XOUT,
                        N := "SIM_DB"."PLANT_DELAY_ACTUAL[Ncycle]",
                        XOUT => "SIM_DB".PLANT_PV_SMITH);
   END_IF;
END_REGION

REGION Network 5: PID目标模型
   RUNG wire#powerrail
      "LAG1_DB_plant_dummy"(RUN := "SIM_DB".SIM_RUN, XIN := "TEST_PID_DB".XOUT, TAU := "SIM_DB"."PLANT_TAU_ACTUAL[ms]", CYCLE := 100.0, XOUT =>)
      "DELAY_DB_plant_dummy"(RUN := "SIM_DB".SIM_RUN, XIN := "LAG1_DB_plant_dummy".XOUT, N := "SIM_DB"."PLANT_DELAY_ACTUAL[Ncycle]", XOUT => "SIM_DB".PLANT_PV_PID)
   END_RUNG
   // the same network as SCL:
   "LAG1_DB_plant_dummy"(RUN := "SIM_DB".SIM_RUN,   // "LAG1"
                         XIN := "TEST_PID_DB".XOUT,
                         TAU := "SIM_DB"."PLANT_TAU_ACTUAL[ms]",
                         CYCLE := 100.0,
                         ENO => #_w1);
   IF #_w1 THEN
       "DELAY_DB_plant_dummy"(RUN := "SIM_DB".SIM_RUN,   // "DELAY"
                              XIN := "LAG1_DB_plant_dummy".XOUT,
                              N := "SIM_DB"."PLANT_DELAY_ACTUAL[Ncycle]",
                              XOUT => "SIM_DB".PLANT_PV_PID);
   END_IF;
END_REGION
END_ORGANIZATION_BLOCK

// ===== library types =====

// folder: 5 Data handling

FUNCTION_BLOCK "LGF_FIFO"   // FB10017, SCL
{ S7_Optimized_Access := 'TRUE' }
   VAR_INPUT
      execute : Bool;   // The instruction is executed when a positive signal edge is detected at the "request" parameter.
      mode : Bool;   // 0 = The first entry in the ring buffer is returned. 1 = An entry is written at the last position in the ring buffer.
      initialValue : Variant;   // Value with which the ARRAY of the ring buffer is initialized.
      resetBuffer : Bool;
   END_VAR
   VAR_OUTPUT
      done : Bool;
      error : Bool;
      statusID : UInt;
      status : Word;   // Status information
   END_VAR
   VAR_IN_OUT
      item : Variant;   // The entry that is either returned from the ring buffer or written to the ring buffer
      buffer : Variant;   // An ARRAY that is used as a ring buffer.
   END_VAR
   VAR
      statEdgeupm : Bool;   // Edge memory bit in which the RLO of the previous query is saved.
      statFirstItemIndex : Int := -1;   // Index of the oldest entry in the ring buffer
      statNextEmptyItemIndex : Int := 0;   // Index of the next free entry in the ring buffer
   END_VAR
   VAR_TEMP
      tempEdgeup : Bool;   // Result of edge evaluation
      tempInternalError : Int;   // Error information
      tempNewFirstItemIndex : Int;   // Variable index
      tempNewNextEmptyItemIndex : Int;   // Variable index
      tempPufferSize : UDInt;   // Number of ARRAY elements in the ring buffer
      tempSizeCounter : Int;
   END_VAR
   VAR CONSTANT
      NO_ERROR : Word := 16#0000;
      NO_CURRENT_JOBS : Word := 16#7000;
      BUFFER_EMPTY : Word := 16#8001;
      BUFFER_FULL : Word := 16#8002;
      NO_ARRAY : Word := 16#8200;
      WRONG_TYPE_1 : Word := 16#8201;
      WRONG_TYPE_2 : Word := 16#8202;
      INDEX_IN_ARRAY_LIMITS_1 : Word;
      INDEX_IN_ARRAY_LIMITS_2 : Word;
      ERROR_IN_THIS_BLOCK : UInt := 1;
      ERROR_MOVE_BLK_VARIANT : UInt := 2;
      NEXT_TASK_TO_EXECUTE : Bool := false;
      BUFFER_IS_EMPTY : Int := -1;
      BUFFER_CONTAINS_ARRAY : Int := 0;
      NO_INTERNAL_ERROR : Int := 0;
      BUFFER_INITIALIZED : Int := -1;
      RESET : Bool := true;
   END_VAR
BEGIN
   //=============================================================================
   // SIEMENS AG
   // (c)Copyright 2017
   //-----------------------------------------------------------------------------
   // Library:       LGF (Library General Functions)
   // Tested with:   CPU1212C DC/DC/DC FW:V4.2
   // Engineering:   TIA Portal V14
   // Restrictions:  -
   // Requirements:  PLC (S7-1200 / S7-1500)
   // Functionality: FIFO(First In First Out)-functionblock
   //-----------------------------------------------------------------------------
   // Change log table:
   // Version  Date        Expert in charge / Changes applied
   // 01.00.00 19.08.2015  Siemens Industry Online Support
   //                      First released version
   // 01.00.01 16.11.2015  Siemens Industry Online Support
   //                      Bug fix resetBuffer
   // 01.00.02 02.01.2017  Siemens Industry Online Support
   //                      Upgrade: TIA Portal V14 Update 1
   //=============================================================================

   //This program code section is only executed once after a negative signal edge.
   IF #execute = false AND #statEdgeupm = true THEN
     #done := false;
     // If no error occurred during program execution, the error code "0000" is output.  
     #error := false;
     #statusID := #ERROR_IN_THIS_BLOCK;
     #status := #NO_CURRENT_JOBS;
   END_IF;

   //This program code section is only executed once after a positive signal edge.
   //IF there is no change in the signal state OF the result OF logic operation,
   //the program processing OF the "FIFOQueue" FB is terminated.

   IF #execute <> true OR #statEdgeupm <> false THEN
     #statEdgeupm := #execute;
     RETURN;
   END_IF;
   #statEdgeupm := #execute;

   // ------Validation of whether all parameter inputs are valid.----

   //This program code section checks whether the ring #buffer is an ARRAY.
   //IF so, the number OF the ARRAY elements is read out.
   //IF it is NOT an ARRAY, the program execution is terminated at this point
   //AND the status code "8200" is output.

   IF NOT (IS_ARRAY(#buffer)) THEN
     #error := true;
     #statusID := #ERROR_IN_THIS_BLOCK;
     #status := #NO_ARRAY;
     RETURN;
   ELSE
     #tempPufferSize := CountOfElements(#buffer);
   END_IF;

   //This program code section checks whether the data type OF the ARRAY elements matches
   //the data type OF the entry (tag #item). IF the data types DO NOT match,
   //the program execution is terminated at this point AND the error code "8201" is output.

   IF NOT (TypeOf(#item) = TypeOfElements(#buffer)) THEN
     #error := true;
     #statusID := #ERROR_IN_THIS_BLOCK;
     #status := #WRONG_TYPE_1;
     RETURN;
   END_IF;

   //This program code section checks whether the initial value OF the ring #buffer
   //matches the entry (tag #item). IF the data types DO NOT match,
   //the program execution is terminated at this point
   //AND the error code "8202" is output. *)

   IF NOT (TypeOf(#item) = TypeOf(#initialValue)) THEN
     #error := true;
     #statusID := #ERROR_IN_THIS_BLOCK;
     #status := #WRONG_TYPE_2;
     RETURN;
   END_IF;

   //This program code section checks whether the variable indices are within the ARRAY limits.
   //IF they are NOT, the program execution is terminated at this point
   //AND either error code "8601" OR "8602" is output depending on the index. *)

   IF (#statNextEmptyItemIndex >= #tempPufferSize) THEN
     #error := true;
     #statusID := #ERROR_IN_THIS_BLOCK;
     #status := #INDEX_IN_ARRAY_LIMITS_1;
     RETURN;
   END_IF;

   IF (#statFirstItemIndex >= #tempPufferSize) THEN
     #error := true;
     #statusID := #ERROR_IN_THIS_BLOCK;
     #status := #INDEX_IN_ARRAY_LIMITS_2;
     RETURN;
   END_IF;


   //If reset is "TRUE" the buffer and their  counters are resetted
   IF #resetBuffer = #RESET THEN
     #statFirstItemIndex := -1;
     #statNextEmptyItemIndex := 0;

     FOR #tempSizeCounter := 0 TO UDINT_TO_INT(#tempPufferSize - 1) DO

       #tempInternalError := MOVE_BLK_VARIANT(SRC := #initialValue,
                                              COUNT := 1,
                                              SRC_INDEX := 0,
                                              DEST_INDEX := #tempSizeCounter,
                                              DEST => #buffer);
     END_FOR;
     IF (#tempInternalError <> #NO_INTERNAL_ERROR) THEN
       #error := true;
       #statusID := #ERROR_MOVE_BLK_VARIANT;
       #status := INT_TO_WORD(#tempInternalError);
     END_IF;
     RETURN;
   END_IF;

   //-----------Program code execution, depending on the Mode parameter-------------
   // The execution of the instructions depends on the signal state of the Mode parameter.

   IF #mode = #NEXT_TASK_TO_EXECUTE THEN


     // If the Mode parameter has the signal state "0",
     // the first entry from the passed ring buffer is returned.

     //this program code section checks whether the ring #buffer is empty.
     //IF this is the CASE, program execution is terminated at this point
     //AND the error code "8001" is output. *)

     IF (#statFirstItemIndex = #BUFFER_IS_EMPTY) THEN
       #error := true;
       #statusID := #ERROR_IN_THIS_BLOCK;
       #status := #BUFFER_EMPTY;
       RETURN;
     END_IF;


     // This program code section returns the first entry of the ring buffer.

     #tempInternalError := MOVE_BLK_VARIANT(SRC := #buffer,
                                            COUNT := 1,
                                            SRC_INDEX := #statFirstItemIndex,
                                            DEST_INDEX := 0,
                                            DEST => #item);

     IF (#tempInternalError = #BUFFER_CONTAINS_ARRAY) THEN

       //This program code section checks whether the ring #buffer contains ARRAY elements.
       //IF it does, the first entry is passed further on
       //AND the index is incremented BY 1. *)

       #tempInternalError := MOVE_BLK_VARIANT(SRC := #initialValue,
                                              COUNT := 1,
                                              SRC_INDEX := 0,
                                              DEST_INDEX := #statFirstItemIndex,
                                              DEST => #buffer);

       // This program code section calculates the new index of the first entry.

       #tempNewFirstItemIndex := #statFirstItemIndex + 1;
       #tempNewFirstItemIndex := #tempNewFirstItemIndex MOD UDINT_TO_INT(#tempPufferSize);

       // This program section checks whether the ring buffer is empty.        
       IF (#statNextEmptyItemIndex = #tempNewFirstItemIndex) THEN
         // If the ring buffer is empty, the index is set to 0.            
         #statFirstItemIndex := -1;
         #statNextEmptyItemIndex := 0;
       ELSE
         // The index of the first entry is changed.            
         #statFirstItemIndex := #tempNewFirstItemIndex;
       END_IF;
     END_IF;
   ELSE

     // If the Mode parameter has the signal state "1", the entry is written to the passed ring buffer.

     //this program code section checks whether the ring #buffer is full.
     //IF this is the CASE, program execution is terminated at this point
     //AND the error code "8002" is output. *)

     IF (#statNextEmptyItemIndex = #statFirstItemIndex) THEN
       #error := true;
       #statusID := #ERROR_IN_THIS_BLOCK;
       #status := #BUFFER_FULL;
       RETURN;
     END_IF;

     // This program code section writes the entry to the ring buffer.   
     #tempInternalError := MOVE_BLK_VARIANT(SRC := #item,
                                            COUNT := 1,
                                            SRC_INDEX := 0,
                                            DEST_INDEX := #statNextEmptyItemIndex,
                                            DEST => #buffer);

     IF (#tempInternalError = #NO_INTERNAL_ERROR) THEN

       // This program code section increments the index by 1 and calculates the new empty entry index.        
       #tempNewNextEmptyItemIndex := #statNextEmptyItemIndex + 1;
       #tempNewNextEmptyItemIndex := #tempNewNextEmptyItemIndex MOD UDINT_TO_INT(#tempPufferSize);
       #statNextEmptyItemIndex := #tempNewNextEmptyItemIndex;

       //This program code section checks which index the "#firstItemIndex" tag has.
       //IF the number = -1, the ring buffer is initialized
       //AND the entry is written TO the ring #buffer.
       //Therefore, "0" must be assigned TO the tag.

       IF (#statFirstItemIndex = #BUFFER_INITIALIZED) THEN
         #statFirstItemIndex := 0;
       END_IF;
     END_IF;
   END_IF;

   //-------------------------Local error handling----------------------------
   //This program code section checks whether a "Local" #error has occurred.
   //IF This is the CASE, program execution is terminated at This point
   //AND the error code of MOV_BLK_VARIANT is output. *)

   IF (#tempInternalError <> #NO_INTERNAL_ERROR) THEN
     #error := true;
     #statusID := #ERROR_MOVE_BLK_VARIANT;
     #status := INT_TO_WORD(#tempInternalError);
     RETURN;
   END_IF;

   #done := true;
   #status := #NO_ERROR;
END_FUNCTION_BLOCK

FUNCTION_BLOCK "LGF_RingBuffer"   // FB10022, SCL
{ S7_Optimized_Access := 'TRUE' }
VERSION : 0.1
   VAR_INPUT
      write : Bool;   // With a rising edge newValue is written in ring buffer
      resetBuffer : Bool;   // Reset buffer
      newValue : Word;   // New Value
   END_VAR
   VAR_IN_OUT
      buffer : Array[*] of Word;   // Buffer
   END_VAR
   VAR
      statInitialized : Bool;   // -
      statElementReset : DInt;   // -
      statLowerLimit : DInt;   // -
      statUpperLimit : DInt;   // -
      statNumElements : UDInt;   // -
      statEdgeWrite : Bool;
   END_VAR
   VAR_TEMP
      tempRetVal : Int;   // -
   END_VAR
BEGIN
   //=============================================================================
   // Siemens AG
   // (c)Copyright 2017
   //-----------------------------------------------------------------------------
   // Library:       LGF (Library General Functions)
   // Tested with:   CPU1212C DC/DC/DC FW:V4.2
   // Engineering:   TIA Portal V14 SP1 Upd 5
   // Restrictions:  -
   // Requirements:  PLC (S7-1200 / S7-1500)
   // Functionality: Ring buffer-functionblock
   //-----------------------------------------------------------------------------
   // Change log table:
   // Version  Date        In charge / Changes applied
   // 01.00.00 03.07.2018  Siemens Industry Online Support
   //                      First released version
   //=============================================================================

   // Initialization
   IF (NOT #statInitialized)
   THEN
     #statLowerLimit := LOWER_BOUND(ARR := #buffer, DIM := 1);
     #statUpperLimit := UPPER_BOUND(ARR := #buffer, DIM := 1);
     #statNumElements := DINT_TO_UDINT(#statUpperLimit - #statLowerLimit + 1);
     #statInitialized := true;
   END_IF;

   IF (#write = TRUE)
     AND (NOT #statEdgeWrite)
     AND (NOT #resetBuffer)
   THEN
     // Move all elements but the last one one element up
     #tempRetVal := MOVE_BLK_VARIANT(SRC := #buffer,
                                     COUNT := #statNumElements - 1,
                                     SRC_INDEX := 0,
                                     DEST_INDEX := 1,
                                     DEST => #buffer);
     // Store new value to first element
     #buffer[#statLowerLimit] := #newValue;
   END_IF;

   IF (#resetBuffer = TRUE)
   THEN
     // Reset buffer
     FOR #statElementReset := #statLowerLimit TO #statUpperLimit DO
       // Statement section FOR
       #buffer[#statElementReset] := 0;
     END_FOR;

   END_IF;

   // Edge detection
   #statEdgeWrite := #write;
END_FUNCTION_BLOCK